TYPE Belt :
STRUCT
	cmd  AT%Q*	: UINT;
	freq AT%Q*	: UINT;
END_STRUCT
END_TYPE

(* stored: Version 1.1.0.1, ProductVersion 3.1.4024.12
   DUT Belt: Id {6625f086-4162-4780-bb7b-f5160f2f835b} *)
